(* PLC project Unnamed, Unknown Unnamed 1 *)
(* stored: creationDateTime 2019-08-06T14:23:42, modificationDateTime 2022-01-18T11:38:21 *)

FUNCTION_BLOCK PumpControl
  VAR_INPUT
    Pump : HMI_NODE := 1;
  END_VAR
  VAR
    Pressure : HMI_INT;
  END_VAR
  VAR_INPUT
    TargetPressure : INT;
  END_VAR
  VAR
    Sloth : HMI_INT;
    boolout : HMI_BOOL;
    boolin : HMI_BOOL := True;
    strout : HMI_STRING;
    strin : HMI_STRING := blup;
    floating : HMI_REAL;
  END_VAR
  VAR  (* added by the conversion: wires and edge detectors of the diagram *)
    _SUB7_OUT : INT;
  END_VAR

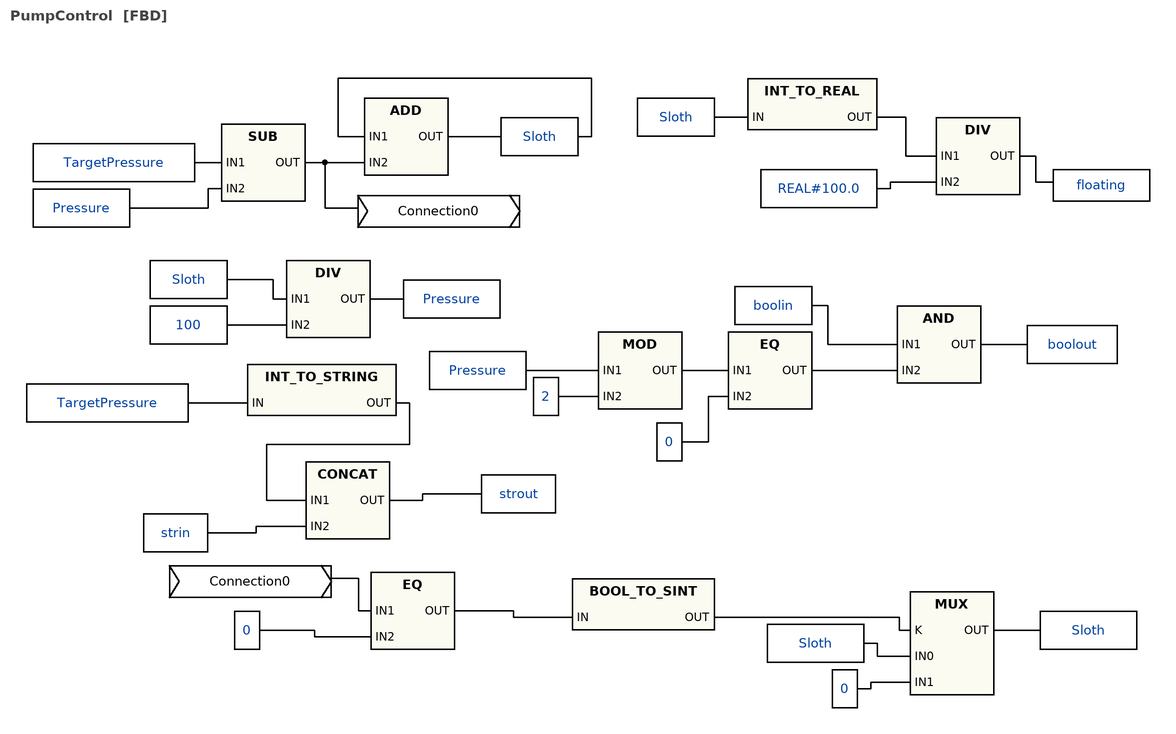
(* FBD diagram, written out as Structured Text *)
_SUB7_OUT := TargetPressure - Pressure;
Sloth := Sloth + _SUB7_OUT;
floating := INT_TO_REAL(Sloth) / REAL#100.0;
Pressure := Sloth / 100;
boolout := boolin AND Pressure MOD 2 = 0;
strout := CONCAT(INT_TO_STRING(TargetPressure), strin);
Sloth := MUX(BOOL_TO_SINT(_SUB7_OUT = 0), Sloth, 0);
END_FUNCTION_BLOCK

PROGRAM MainStuff
  VAR
    TargetPressure : HMI_INT;
    selection : HMI_INT;
    Pump0 : PumpControl;
    Pump1 : PumpControl;
    Pump2 : PumpControl;
    Pump3 : PumpControl;
    Pump4 : PumpControl;
    Pump5 : PumpControl;
    Pump6 : PumpControl;
    Pump7 : PumpControl;
  END_VAR
  VAR_EXTERNAL
    CURRENT_PAGE_0 : HMI_STRING;
  END_VAR
  VAR
    PAGESWITCH : BOOL;
    R_TRIG0 : R_TRIG;
  END_VAR

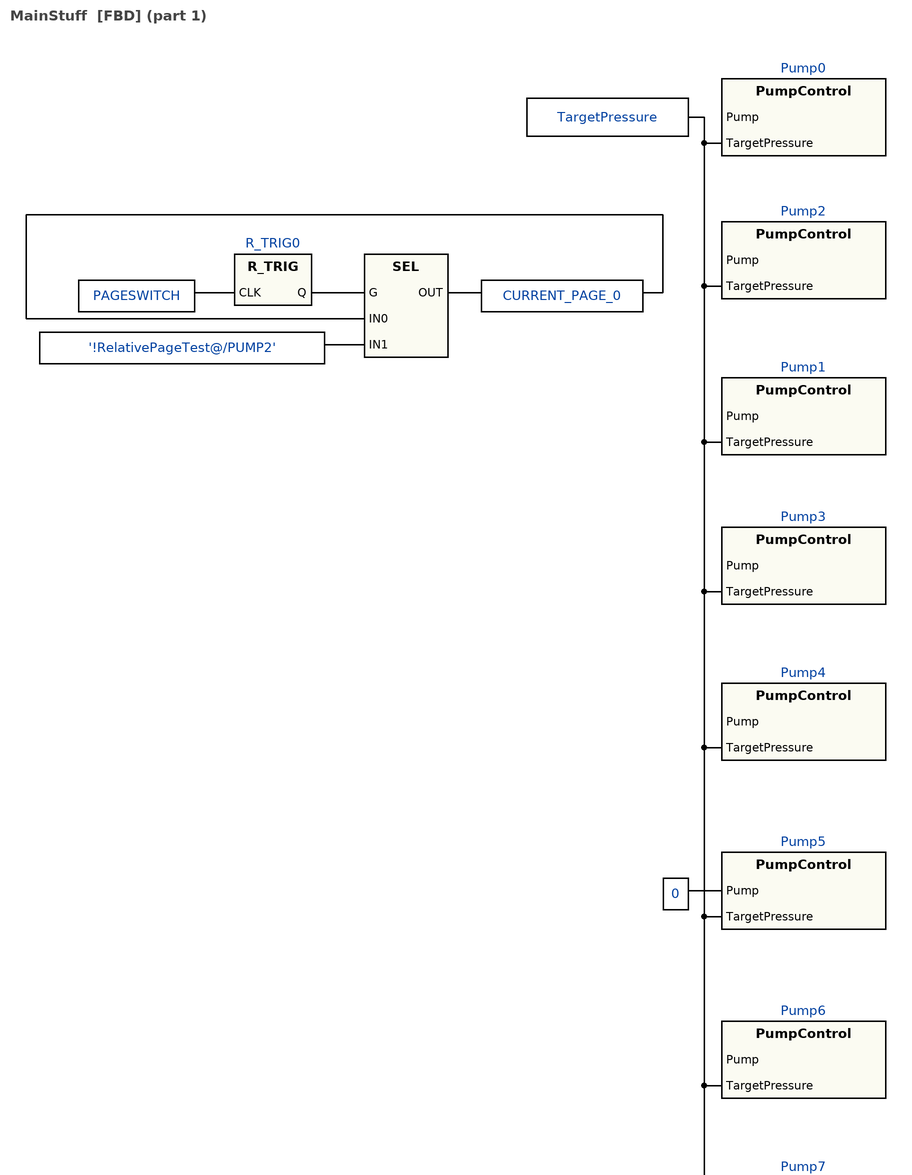
(* FBD diagram, written out as Structured Text *)
R_TRIG0(CLK := PAGESWITCH);
CURRENT_PAGE_0 := SEL(R_TRIG0.Q, CURRENT_PAGE_0, '!RelativePageTest@/PUMP2');
Pump0(TargetPressure := TargetPressure);
Pump2(TargetPressure := TargetPressure);
Pump1(TargetPressure := TargetPressure);
Pump3(TargetPressure := TargetPressure);
Pump4(TargetPressure := TargetPressure);
Pump5(Pump := 0, TargetPressure := TargetPressure);
Pump6(TargetPressure := TargetPressure);
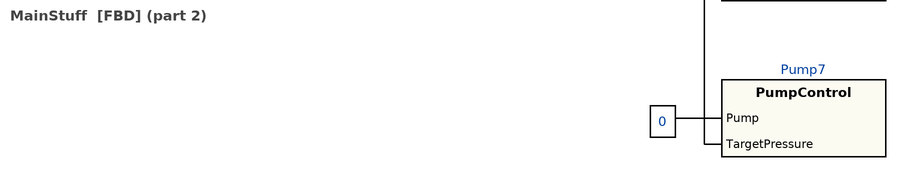
Pump7(Pump := 0, TargetPressure := TargetPressure);
END_PROGRAM

CONFIGURATION config
  RESOURCE resource1 ON PLC
    TASK task0(INTERVAL := T#20ms, PRIORITY := 0);
    PROGRAM instance0 WITH task0 : MainStuff;
  END_RESOURCE
END_CONFIGURATION
